(* This function block is created for interface devices between different PLC*)
(* Not all the Variables in the original structure is required, just few signals *)
(* They have to be linked to the custom created variables on the EL6692/5 primary side*)
FUNCTION_BLOCK FB_Gauge_Interface
VAR_INPUT
END_VAR
VAR_OUTPUT
	{attribute 'pytmc' := 'pv:'}
	VG : ST_VG;
END_VAR
VAR
	i_rPRESS AT%I*: REAL;  //This is the human-readable pressure
	i_xAT_VAC AT%I*: BOOL;
	i_xPRESS_OK AT%I*: BOOL;
	
END_VAR

(* This function block is created for interface devices between different PLC*)
(* Not all the Variables in the original structure is required, just few signals *)
(* They have to be linked to the custom created variables on the EL6692/5 primary side*)

VG.rPRESS := i_rPRESS;
VG.xAT_VAC := i_xAT_VAC;
VG.xPRESS_OK := i_xPRESS_OK;

END_FUNCTION_BLOCK

(* stored: Version 1.1.0.1, ProductVersion 3.1.4022.16
   POU FB_Gauge_Interface: Id {1ed0a657-4e26-4a4b-9434-968a1918180c}, SpecialFunc None *)
